// TwinCAT 3 PLC project PLCStudent
// ProgramVersion: 3.1.4022.3
// libraries:
//   Tc2_Standard, * (Beckhoff Automation GmbH)
//   Tc2_System, * (Beckhoff Automation GmbH)
//   Tc3_Module, * (Beckhoff Automation GmbH)
// project tree:
//   GVLs/ GVL.TcGVL (not stored)
//   / PlcTask.TcTTO (not stored)
//   POUs/ BtnRequestFBD.TcPOU, ControlElvSFC.TcPOU, ControlLD.TcPOU, ControlQ_LD.TcPOU, InQ.TcPOU, MAIN.TcPOU, QueueSTFBD.TcPOU
// (motion and I/O tree: see PLC project plcsim)
// real-time tasks:
//   TASK PlcTask: cycle T#20ms, priority 20, ADS port 350
// variable links:
//   PLCSim/PLCSim Instance <-> PLCStudent/PLCStudent Instance
//     PlcTask Inputs/GVL.iiDisplayElevat <-> PlcTask Outputs/GVL.qiDispElevat
//     PlcTask Inputs/GVL.ixDoorClose <-> PlcTask Outputs/GVL.qxDoorClose
//     PlcTask Inputs/GVL.ixLampElevat1 <-> PlcTask Outputs/GVL.qxLampElevat1
//     PlcTask Inputs/GVL.ixLampElevat2 <-> PlcTask Outputs/GVL.qxLampElevat2
//     PlcTask Inputs/GVL.ixLampElevat3 <-> PlcTask Outputs/GVL.qxLampElevat3
//     PlcTask Inputs/GVL.ixLampLevel1 <-> PlcTask Outputs/GVL.qxLampLevel1
//     PlcTask Inputs/GVL.ixLampLevel2 <-> PlcTask Outputs/GVL.qxLampLevel2
//     PlcTask Inputs/GVL.ixLampLevel3 <-> PlcTask Outputs/GVL.qxLampLevel3
//     PlcTask Inputs/GVL.ixMotorDown <-> PlcTask Outputs/GVL.qxMotorDown
//     PlcTask Inputs/GVL.ixMotorUp <-> PlcTask Outputs/GVL.qxMotorUp
//     PlcTask Outputs/GVL.qxButtElevat1 <-> PlcTask Inputs/GVL.ixButtElevat1
//     PlcTask Outputs/GVL.qxButtElevat2 <-> PlcTask Inputs/GVL.ixButtElevat2
//     PlcTask Outputs/GVL.qxButtElevat3 <-> PlcTask Inputs/GVL.ixButtElevat3
//     PlcTask Outputs/GVL.qxButtGreen <-> PlcTask Inputs/GVL.ixButtGreen
//     PlcTask Outputs/GVL.qxButtLevel1 <-> PlcTask Inputs/GVL.ixButtLevel1
//     PlcTask Outputs/GVL.qxButtLevel2 <-> PlcTask Inputs/GVL.ixButtLevel2
//     PlcTask Outputs/GVL.qxButtLevel3 <-> PlcTask Inputs/GVL.ixButtLevel3
//     PlcTask Outputs/GVL.qxButtRed <-> PlcTask Inputs/GVL.ixButtRed
//     PlcTask Outputs/GVL.qxDoorClosed <-> PlcTask Inputs/GVL.ixDoorClosed
//     PlcTask Outputs/GVL.qxDoorOpen <-> PlcTask Inputs/GVL.ixDoorOpen
//     PlcTask Outputs/GVL.qxElevatLevel1 <-> PlcTask Inputs/GVL.ixElevatLevel1
//     PlcTask Outputs/GVL.qxElevatLevel2 <-> PlcTask Inputs/GVL.ixElevatLevel2
//     PlcTask Outputs/GVL.qxElevatLevel3 <-> PlcTask Inputs/GVL.ixElevatLevel3

// ---- POUs/BtnRequestFBD.TcPOU
FUNCTION_BLOCK BtnRequestFBD
VAR_INPUT
	ixButtonElevat1 : BOOL ;
	ixButtonLevel1 : BOOL ;
	ixButtonElevat2 : BOOL ;
	ixButtonLevel2 : BOOL ;
	ixButtonElevat3 : BOOL ;
	ixButtonLevel3 : BOOL ;
END_VAR
VAR_OUTPUT
	ixQueue : BOOL ;
	iiQueueOrder : INT ;
END_VAR
VAR
END_VAR

IF ixButtonElevat1 OR ixButtonLevel1 THEN
	iiQueueOrder := 1 ;
	ixQueue := TRUE ;
ELSIF ixButtonElevat2 OR ixButtonLevel2 THEN
	iiQueueOrder := 2 ;
	ixQueue := TRUE ;
ELSIF ixButtonElevat3 OR ixButtonLevel3 THEN
	iiQueueOrder := 3 ;
	ixQueue := TRUE ;
ELSE
	iiQueueOrder := - 1 ;
	ixQueue := FALSE ;
END_IF

END_FUNCTION_BLOCK

// ---- POUs/ControlElvSFC.TcPOU
PROGRAM ControlElvSFC
VAR
	SendDequeue: INT;
	ResetDequeue: BOOL;
	SendDequeue1: BOOL;
	Reset: INT;
	ResetDequeue_1: BOOL;
	SendDequeue2: BOOL;
	ResetDequeue_2: BOOL;
	SendDequeue3: BOOL;
	ResetDequeue_3: BOOL;
END_VAR

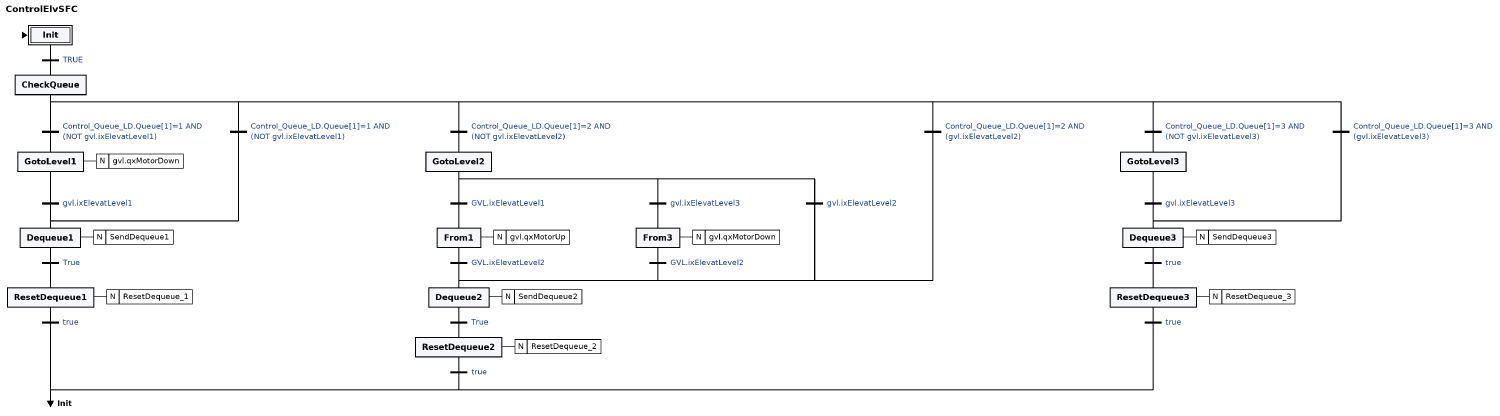
INITIAL_STEP Init:
END_STEP
TRANSITION FROM Init TO CheckQueue
    := TRUE;
END_TRANSITION
STEP CheckQueue:
END_STEP
TRANSITION FROM CheckQueue TO GotoLevel1
    := Control_Queue_LD.Queue[1]=1 AND (NOT gvl.ixElevatLevel1);
END_TRANSITION
STEP GotoLevel1:
    gvl.qxMotorDown(N);
END_STEP
TRANSITION FROM GotoLevel1 TO Dequeue1
    := gvl.ixElevatLevel1;
END_TRANSITION
TRANSITION FROM CheckQueue TO Dequeue1
    := Control_Queue_LD.Queue[1]=1 AND (NOT gvl.ixElevatLevel1);
END_TRANSITION
STEP Dequeue1:
    SendDequeue1(N);
END_STEP
TRANSITION FROM Dequeue1 TO ResetDequeue1
    := True;
END_TRANSITION
STEP ResetDequeue1:
    ResetDequeue_1(N);
END_STEP
TRANSITION FROM ResetDequeue1 TO Init
    := true;
END_TRANSITION
TRANSITION FROM CheckQueue TO GotoLevel2
    := Control_Queue_LD.Queue[1]=2 AND (NOT gvl.ixElevatLevel2);
END_TRANSITION
STEP GotoLevel2:
END_STEP
TRANSITION FROM GotoLevel2 TO From1
    := GVL.ixElevatLevel1;
END_TRANSITION
STEP From1:
    gvl.qxMotorUp(N);
END_STEP
TRANSITION FROM From1 TO Dequeue2
    := GVL.ixElevatLevel2;
END_TRANSITION
TRANSITION FROM GotoLevel2 TO From3
    := gvl.ixElevatLevel3;
END_TRANSITION
STEP From3:
    gvl.qxMotorDown(N);
END_STEP
TRANSITION FROM From3 TO Dequeue2
    := GVL.ixElevatLevel2;
END_TRANSITION
TRANSITION FROM GotoLevel2 TO Dequeue2
    := gvl.ixElevatLevel2;
END_TRANSITION
TRANSITION FROM CheckQueue TO Dequeue2
    := Control_Queue_LD.Queue[1]=2 AND (gvl.ixElevatLevel2);
END_TRANSITION
STEP Dequeue2:
    SendDequeue2(N);
END_STEP
TRANSITION FROM Dequeue2 TO ResetDequeue2
    := True;
END_TRANSITION
STEP ResetDequeue2:
    ResetDequeue_2(N);
END_STEP
TRANSITION FROM ResetDequeue2 TO Init
    := true;
END_TRANSITION
TRANSITION FROM CheckQueue TO GotoLevel3
    := Control_Queue_LD.Queue[1]=3 AND (NOT gvl.ixElevatLevel3);
END_TRANSITION
STEP GotoLevel3:
END_STEP
TRANSITION FROM GotoLevel3 TO Dequeue3
    := gvl.ixElevatLevel3;
END_TRANSITION
TRANSITION FROM CheckQueue TO Dequeue3
    := Control_Queue_LD.Queue[1]=3 AND (gvl.ixElevatLevel3);
END_TRANSITION
STEP Dequeue3:
    SendDequeue3(N);
END_STEP
TRANSITION FROM Dequeue3 TO ResetDequeue3
    := true;
END_TRANSITION
STEP ResetDequeue3:
    ResetDequeue_3(N);
END_STEP
TRANSITION FROM ResetDequeue3 TO Init
    := true;
END_TRANSITION

END_PROGRAM

// ---- POUs/ControlLD.TcPOU
PROGRAM ControlLD
VAR
	Ready: RS;
	level1: RS;
	L1toL3: RS;
	Level3: RS;
	L3ToL1: RS;
	L1toL2: RS;
	L3toL2: RS;
	Level2: RS;
	L2toL1: RS;
	L2toL3: RS;
	MotorUpTimerr: TON;
	MotorDownTimerr: TON;
END_VAR
VAR // added by the converter: edge detectors and wires of the graphical bodies
    _w1, _w2, _w3 : BOOL;
END_VAR

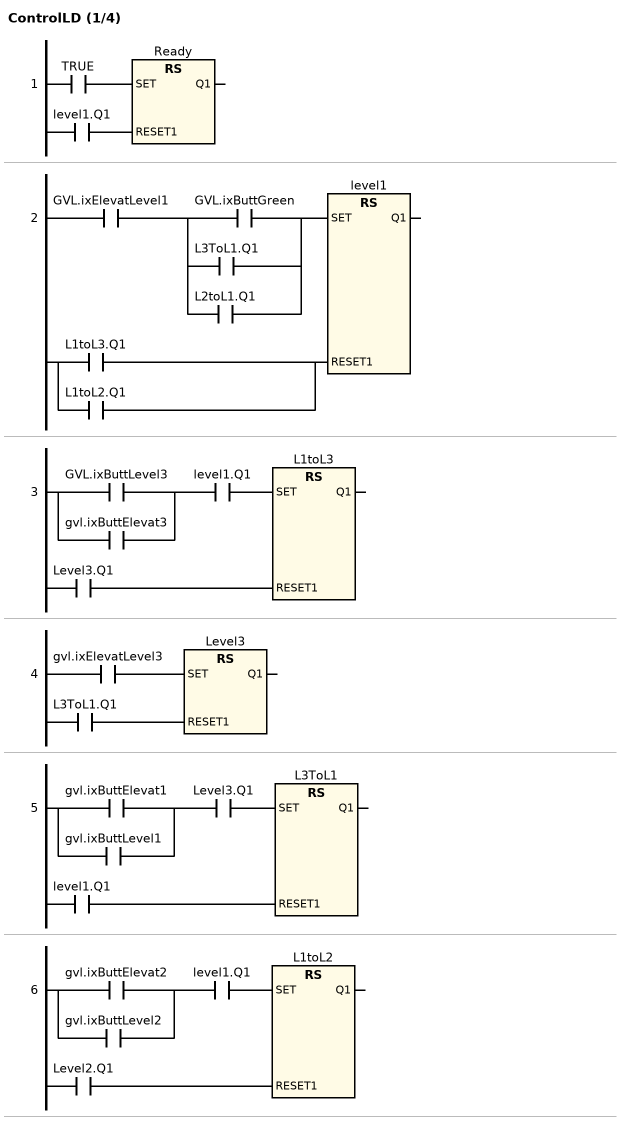
// NETWORK 1
Ready(SET := TRUE, RESET1 := level1.Q1); // RS

// NETWORK 2
level1(SET := GVL.ixElevatLevel1 AND (GVL.ixButtGreen OR L3ToL1.Q1 OR L2toL1.Q1), RESET1 := L1toL3.Q1 OR L1toL2.Q1); // RS

// NETWORK 3
L1toL3(SET := (GVL.ixButtLevel3 OR gvl.ixButtElevat3) AND level1.Q1, RESET1 := Level3.Q1); // RS

// NETWORK 4
Level3(SET := gvl.ixElevatLevel3, RESET1 := L3ToL1.Q1); // RS

// NETWORK 5
L3ToL1(SET := (gvl.ixButtElevat1 OR gvl.ixButtLevel1) AND Level3.Q1, RESET1 := level1.Q1); // RS

// NETWORK 6
L1toL2(SET := (gvl.ixButtElevat2 OR gvl.ixButtLevel2) AND level1.Q1, RESET1 := Level2.Q1); // RS

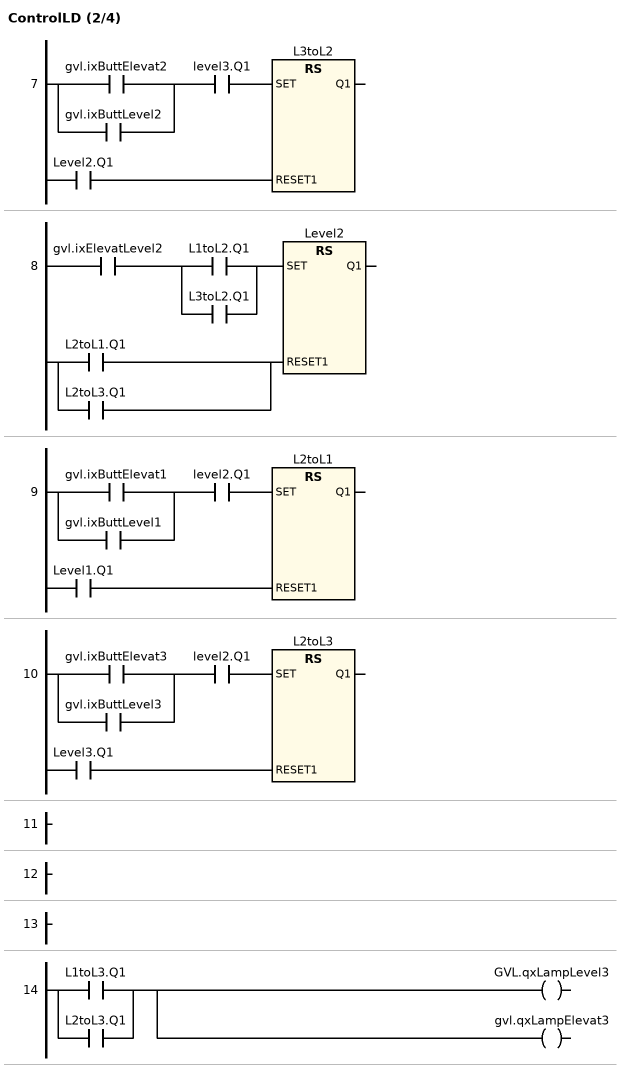
// NETWORK 7
L3toL2(SET := (gvl.ixButtElevat2 OR gvl.ixButtLevel2) AND level3.Q1, RESET1 := Level2.Q1); // RS

// NETWORK 8
Level2(SET := gvl.ixElevatLevel2 AND (L1toL2.Q1 OR L3toL2.Q1), RESET1 := L2toL1.Q1 OR L2toL3.Q1); // RS

// NETWORK 9
L2toL1(SET := (gvl.ixButtElevat1 OR gvl.ixButtLevel1) AND level2.Q1, RESET1 := Level1.Q1); // RS

// NETWORK 10
L2toL3(SET := (gvl.ixButtElevat3 OR gvl.ixButtLevel3) AND level2.Q1, RESET1 := Level3.Q1); // RS

// NETWORK 11

// NETWORK 12

// NETWORK 13

// NETWORK 14
_w1 := L1toL3.Q1 OR L2toL3.Q1;
GVL.qxLampLevel3 := _w1;
gvl.qxLampElevat3 := _w1;

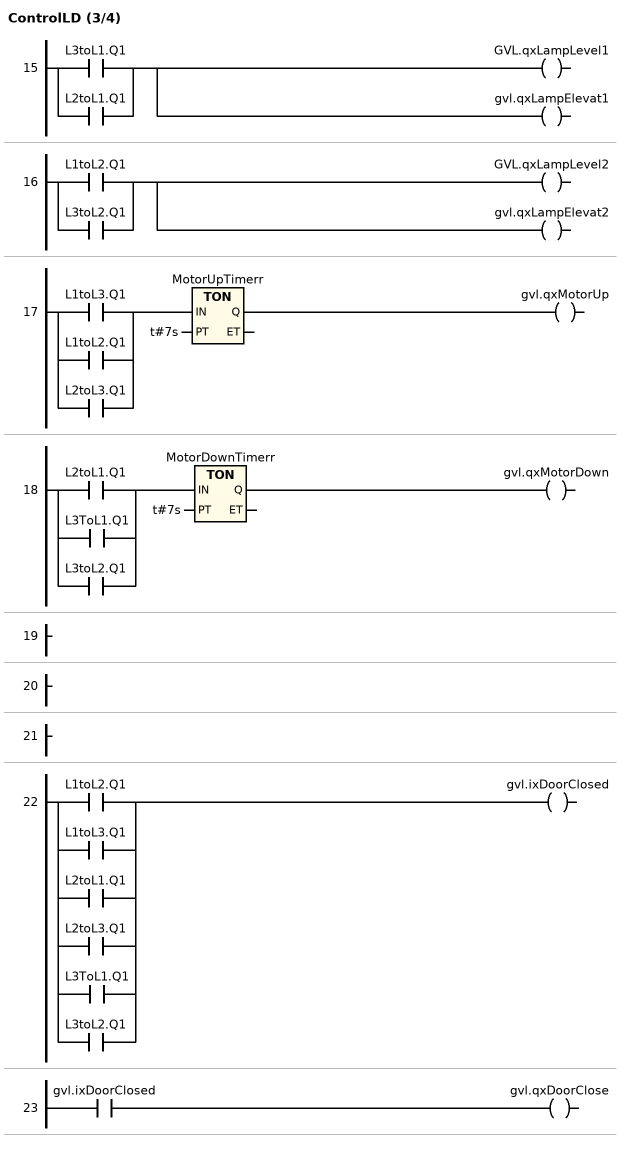
// NETWORK 15
_w2 := L3toL1.Q1 OR L2toL1.Q1;
GVL.qxLampLevel1 := _w2;
gvl.qxLampElevat1 := _w2;

// NETWORK 16
_w3 := L1toL2.Q1 OR L3toL2.Q1;
GVL.qxLampLevel2 := _w3;
gvl.qxLampElevat2 := _w3;

// NETWORK 17
MotorUpTimerr(IN := L1toL3.Q1 OR L1toL2.Q1 OR L2toL3.Q1, PT := t#7s); // TON
gvl.qxMotorUp := MotorUpTimerr.Q;

// NETWORK 18
MotorDownTimerr(IN := L2toL1.Q1 OR L3ToL1.Q1 OR L3toL2.Q1, PT := t#7s); // TON
gvl.qxMotorDown := MotorDownTimerr.Q;

// NETWORK 19

// NETWORK 20

// NETWORK 21

// NETWORK 22
gvl.ixDoorClosed := L1toL2.Q1 OR L1toL3.Q1 OR L2toL1.Q1 OR L2toL3.Q1 OR L3ToL1.Q1 OR L3toL2.Q1;

// NETWORK 23
gvl.qxDoorClose := gvl.ixDoorClosed;

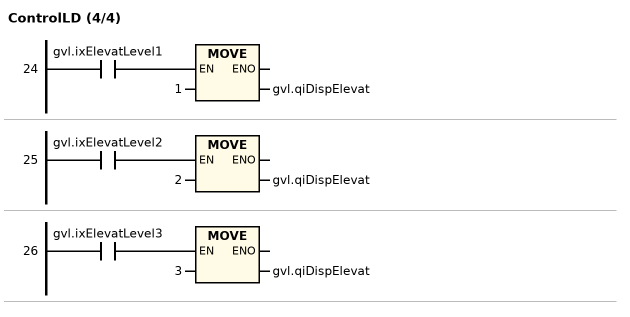
// NETWORK 24
IF gvl.ixElevatLevel1 THEN gvl.qiDispElevat := 1; END_IF

// NETWORK 25
IF gvl.ixElevatLevel2 THEN gvl.qiDispElevat := 2; END_IF

// NETWORK 26
IF gvl.ixElevatLevel3 THEN gvl.qiDispElevat := 3; END_IF

END_PROGRAM

// ---- POUs/ControlQ_LD.TcPOU
PROGRAM ControlQ_LD
VAR
    QueueSTFBD_0 : QueueSTFBD;
    mxQueue : BOOL;
    miOrderQueue : INT;
    Queue : ARRAY [1..3] OF INT;
    ButtonRequstFBD_0 : ButtonRequstFBD;
	QueueSTFBD_2: QueueSTFBD;
	QueueSTFBD_1: QueueSTFBD;
END_VAR
VAR_INPUT
    ixDequeue : BOOL;
    iiOrderDequeue : INT;
END_VAR

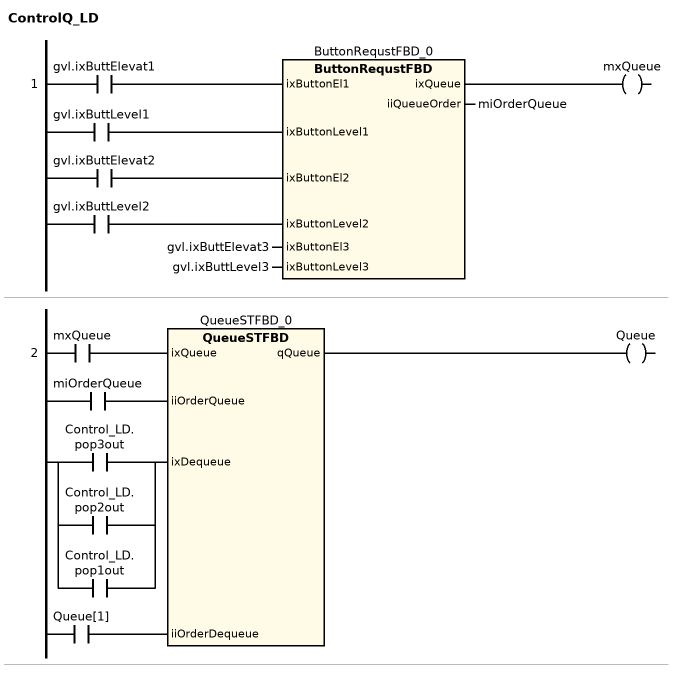
// NETWORK 1
ButtonRequstFBD_0(
    ixButtonEl1 := gvl.ixButtElevat1,
    ixButtonLevel1 := gvl.ixButtLevel1,
    ixButtonEl2 := gvl.ixButtElevat2,
    ixButtonLevel2 := gvl.ixButtLevel2,
    ixButtonEl3 := gvl.ixButtElevat3,
    ixButtonLevel3 := gvl.ixButtLevel3,
    iiQueueOrder => miOrderQueue); // ButtonRequstFBD
mxQueue := ButtonRequstFBD_0.ixQueue;

// NETWORK 2
QueueSTFBD_0(
    ixQueue := mxQueue,
    iiOrderQueue := miOrderQueue,
    ixDequeue := Control_LD.pop3out OR Control_LD.pop2out OR Control_LD.pop1out,
    iiOrderDequeue := Queue[1]); // QueueSTFBD
Queue := QueueSTFBD_0.qQueue;

END_PROGRAM

// ---- POUs/QueueSTFBD.TcPOU
FUNCTION_BLOCK QueueSTFBD
VAR_INPUT
	ixQueue : BOOL ;
	iiOrderQueue : INT ;
	ixDequeue : BOOL ;
	iiOrderDequeue : INT ;
END_VAR
VAR_OUTPUT
	qQueue : ARRAY [ 1 .. 3 ] OF INT := [ 0 , 0 , 0 ] ;
END_VAR
VAR
	State : INT ;
END_VAR

CASE State OF
	0 :
		IF ixQueue AND ( NOT InQueue ( iiNum := iiOrderQueue , iaQueue :=
qQueue ) ) THEN
			State := 1 ;
		END_IF
		IF ixDeQueue AND qQueue [ 1 ] = iiOrderDequeue AND ( NOT ixQueue )
THEN
			State := 2 ;
		END_IF

	1 :
		//DO QUEUE
		IF qQueue [ 1 ] = 0 THEN
			qQueue [ 1 ] := iiOrderQueue ;
		ELSIF qQueue [ 2 ] = 0 THEN
			qQueue [ 2 ] := iiOrderQueue ;
		ELSIF qQueue [ 3 ] = 0 THEN
			qQueue [ 3 ] := iiOrderQueue ;
		END_IF
		State := 0 ;
	2 :
		//DO DEQUEUE
		qQueue [ 1 ] := qQueue [ 2 ] ;
		qQueue [ 2 ] := qQueue [ 3 ] ;
		qQueue [ 3 ] := 0 ;
		State := 0 ;
END_CASE

END_FUNCTION_BLOCK

// ---- POUs/InQ.TcPOU
FUNCTION InQ : BOOL
VAR_INPUT
	iiNum: INT;
	iaQueue:ARRAY[1..3] OF INT;
END_VAR
VAR
END_VAR


IF iiNum=iaQueue[1] OR iiNum=iaQueue[2] OR iiNum=iaQueue[3] THEN
	InQueue:=TRUE;
ELSE
	InQueue:=FALSE;	
END_IF

END_FUNCTION

// ---- POUs/MAIN.TcPOU
PROGRAM MAIN
VAR
END_VAR

Control_LD();

END_PROGRAM
